// TIA Portal project "ScambioFerroviario" (V15.1)

(* hardware
DEVICE "S7-1200 station_1"  S7-1200 Station
   slot 0: "Telaio di montaggio_0"  S7-1200 Rack  Rack  V1.0
   slot 1: "PLC_1"  CPU 1214C DC/DC/DC  6ES7 214-1AG40-0XB0  V4.2
*)

// ===== PLC "PLC_1"  CPU 1214C DC/DC/DC =====

VAR_GLOBAL   // PLC tag table "Tabella delle variabili standard"
   "Mutex" AT %M0.0 : Bool;
   "P1" AT %I0.0 : Bool;
   "P2" AT %I0.1 : Bool;
   "SP1" AT %I0.2 : Bool;
   "SP2" AT %I0.3 : Bool;
   "SA1" AT %I0.4 : Bool;
   "SA2" AT %I0.5 : Bool;
   "A" AT %I0.6 : Bool;
   "B" AT %I0.7 : Bool;
   "C" AT %I1.0 : Bool;
   "D" AT %I1.1 : Bool;
   "S1" AT %Q0.0 : Bool;
   "D1" AT %Q0.1 : Bool;
   "S2" AT %Q0.2 : Bool;
   "D2" AT %Q0.3 : Bool;
   "SC1" AT %Q0.4 : Bool;
   "SC2" AT %Q0.5 : Bool;
END_VAR

VAR_GLOBAL CONSTANT   // PLC tag table "Tabella delle variabili standard"
   "AttesaRifornimento" : Time := T#1m;
END_VAR

TYPE "StatoCorsaSingola"
   STRUCT
      Home : Bool := true;
      Checkpoint : Bool;
      AcquisisciLock : Bool;
      ZonaCritica : Bool;
      RilasciaLock : Bool;
      FineCorsa : Bool;
   END_STRUCT;
END_TYPE

DATA_BLOCK "AndataCarrello1_DB"   // DB1
{ S7_Optimized_Access := 'TRUE' }
VERSION : 0.1
// stored: InstanceOfName CorsaSingola
"CorsaSingola"
BEGIN
END_DATA_BLOCK

DATA_BLOCK "RitornoCarrello1_DB"   // DB2
{ S7_Optimized_Access := 'TRUE' }
VERSION : 0.1
// stored: InstanceOfName CorsaSingola
"CorsaSingola"
BEGIN
END_DATA_BLOCK

DATA_BLOCK "AndataCarrello2_DB"   // DB4
{ S7_Optimized_Access := 'TRUE' }
VERSION : 0.1
// stored: InstanceOfName CorsaSingola
"CorsaSingola"
BEGIN
END_DATA_BLOCK

DATA_BLOCK "RitornoCarrello2_DB"   // DB5
{ S7_Optimized_Access := 'TRUE' }
VERSION : 0.1
// stored: InstanceOfName CorsaSingola
"CorsaSingola"
BEGIN
END_DATA_BLOCK

// folder: System blocks/Program resources

DATA_BLOCK "IEC_Timer_0_DB"   // DB3
{ S7_Optimized_Access := 'TRUE' }
AUTHOR : Simatic
FAMILY : IEC
NAME : IEC_TMR
VERSION : 1.0
// stored: InstanceOfName IEC_TIMER
"IEC_TIMER"
BEGIN
END_DATA_BLOCK

DATA_BLOCK "IEC_Timer_1_DB"   // DB6
{ S7_Optimized_Access := 'TRUE' }
AUTHOR : Simatic
FAMILY : IEC
NAME : IEC_TMR
VERSION : 1.0
// stored: InstanceOfName IEC_TIMER
"IEC_TIMER"
BEGIN
END_DATA_BLOCK

// folder: (top level)

FUNCTION_BLOCK "CorsaSingola"   // FB1, LAD
{ S7_Optimized_Access := 'TRUE' }
VERSION : 0.1
   VAR_INPUT
      Abilita : Bool;
      SP : Bool;
      Fotocellula1 : Bool;
      Fotocellula2 : Bool;
      SA : Bool;
   END_VAR
   VAR_OUTPUT
      SC_0 : Bool;   // Passare qui lo scambio da settare a LOW
      SC_1 : Bool;   // Passare qui lo scambio da settare a HIGH
      "M" : Bool;
   END_VAR
   VAR_IN_OUT
      Mutex : Bool;
   END_VAR
   VAR RETAIN
      Stato : "StatoCorsaSingola";
   END_VAR
BEGIN

REGION Network 1
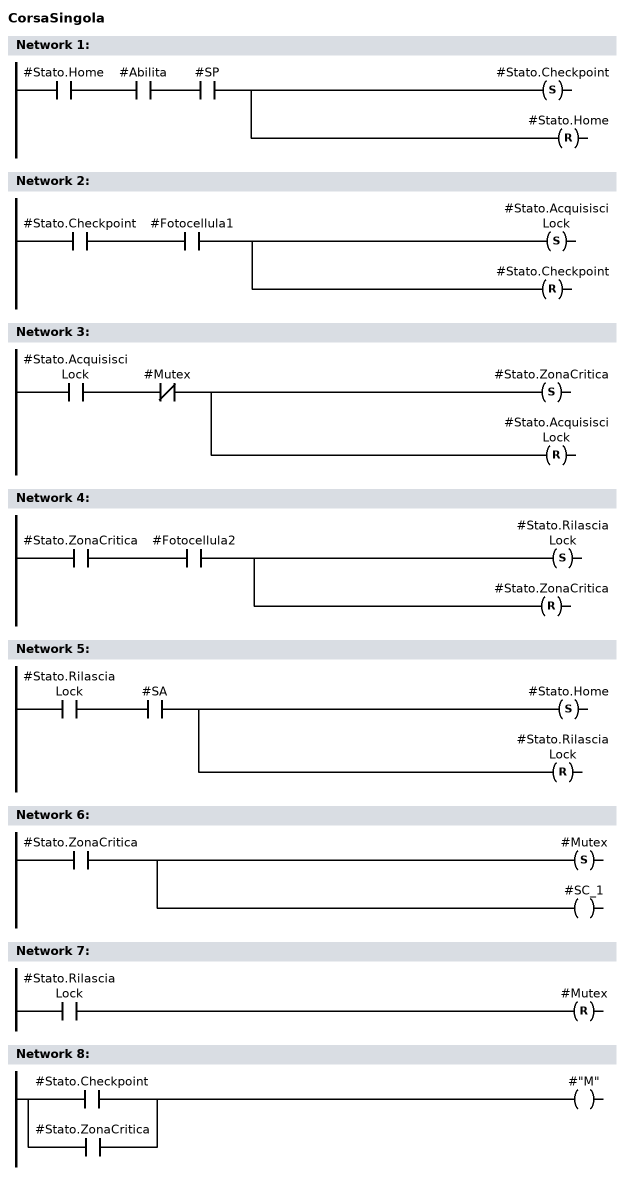
   RUNG wire#powerrail
      Contact( #Stato.Home )
      Contact( #Abilita )
      Contact( #SP )
      wire#w1
      S_Coil( #Stato.Checkpoint )
   END_RUNG
   RUNG wire#w1
      R_Coil( #Stato.Home )
   END_RUNG
   // the same network as SCL:
   IF #Stato.Home AND #Abilita AND #SP THEN
       #Stato.Checkpoint := TRUE;
       #Stato.Home := FALSE;
   END_IF;
END_REGION

REGION Network 2
   RUNG wire#powerrail
      Contact( #Stato.Checkpoint )
      Contact( #Fotocellula1 )
      wire#w1
      S_Coil( #Stato.AcquisisciLock )
   END_RUNG
   RUNG wire#w1
      R_Coil( #Stato.Checkpoint )
   END_RUNG
   // the same network as SCL:
   IF #Stato.Checkpoint AND #Fotocellula1 THEN
       #Stato.AcquisisciLock := TRUE;
       #Stato.Checkpoint := FALSE;
   END_IF;
END_REGION

REGION Network 3
   RUNG wire#powerrail
      Contact( #Stato.AcquisisciLock )
      I_Contact( #Mutex )
      wire#w1
      S_Coil( #Stato.ZonaCritica )
   END_RUNG
   RUNG wire#w1
      R_Coil( #Stato.AcquisisciLock )
   END_RUNG
   // the same network as SCL:
   IF #Stato.AcquisisciLock AND NOT #Mutex THEN
       #Stato.ZonaCritica := TRUE;
       #Stato.AcquisisciLock := FALSE;
   END_IF;
END_REGION

REGION Network 4
   RUNG wire#powerrail
      Contact( #Stato.ZonaCritica )
      Contact( #Fotocellula2 )
      wire#w1
      S_Coil( #Stato.RilasciaLock )
   END_RUNG
   RUNG wire#w1
      R_Coil( #Stato.ZonaCritica )
   END_RUNG
   // the same network as SCL:
   IF #Stato.ZonaCritica AND #Fotocellula2 THEN
       #Stato.RilasciaLock := TRUE;
       #Stato.ZonaCritica := FALSE;
   END_IF;
END_REGION

REGION Network 5
   RUNG wire#powerrail
      Contact( #Stato.RilasciaLock )
      Contact( #SA )
      wire#w1
      S_Coil( #Stato.Home )
   END_RUNG
   RUNG wire#w1
      R_Coil( #Stato.RilasciaLock )
   END_RUNG
   // the same network as SCL:
   IF #Stato.RilasciaLock AND #SA THEN
       #Stato.Home := TRUE;
       #Stato.RilasciaLock := FALSE;
   END_IF;
END_REGION

REGION Network 6
   RUNG wire#powerrail
      Contact( #Stato.ZonaCritica )
      wire#w1
      S_Coil( #Mutex )
   END_RUNG
   RUNG wire#w1
      Coil( #SC_1 )
   END_RUNG
   // the same network as SCL:
   IF #Stato.ZonaCritica THEN #Mutex := TRUE; END_IF;
   #SC_1 := #Stato.ZonaCritica;
END_REGION

REGION Network 7
   RUNG wire#powerrail
      Contact( #Stato.RilasciaLock )
      R_Coil( #Mutex )
   END_RUNG
   // the same network as SCL:
   IF #Stato.RilasciaLock THEN #Mutex := FALSE; END_IF;
END_REGION

REGION Network 8
   RUNG wire#powerrail
      Contact( #Stato.Checkpoint )
      wire#w1
      Coil( #"M" )
   END_RUNG
   RUNG wire#powerrail
      Contact( #Stato.ZonaCritica )
   END_RUNG wire#w1
   // the same network as SCL:
   #"M" := #Stato.Checkpoint OR #Stato.ZonaCritica;
END_REGION
END_FUNCTION_BLOCK

ORGANIZATION_BLOCK "Main"   // OB1, LAD, ProgramCycle
TITLE = "Main Program Sweep (Cycle)"
{ S7_Optimized_Access := 'TRUE' }
VERSION : 0.1
   VAR_INPUT
      Initial_Call : Bool;   // Initial call of this OB
      Remanence : Bool;   // =True, if remanent data are available
   END_VAR
BEGIN

REGION Network 1
   // Carrello1
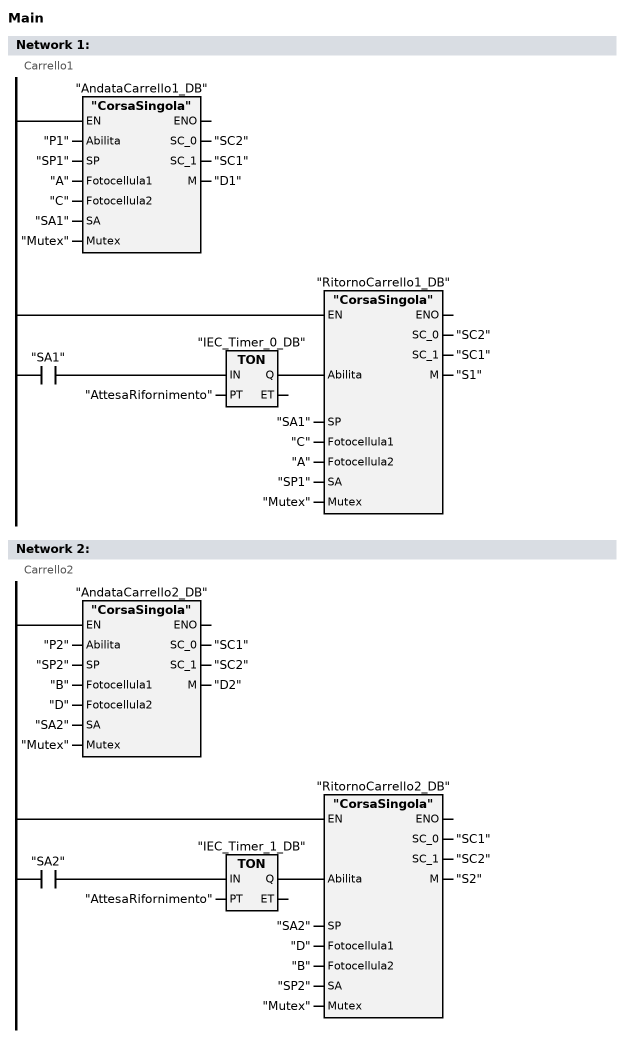
   "AndataCarrello1_DB"(Abilita := "P1",   // "CorsaSingola"
                        SP := "SP1",
                        Fotocellula1 := "A",
                        Fotocellula2 := "C",
                        SA := "SA1",
                        Mutex := "Mutex",
                        SC_0 => "SC2",
                        SC_1 => "SC1",
                        "M" => "D1");
   "IEC_Timer_0_DB".TON(IN := "SA1", PT := "AttesaRifornimento");
   "RitornoCarrello1_DB"(Abilita := "IEC_Timer_0_DB".Q,   // "CorsaSingola"
                         SP := "SA1",
                         Fotocellula1 := "C",
                         Fotocellula2 := "A",
                         SA := "SP1",
                         Mutex := "Mutex",
                         SC_0 => "SC2",
                         SC_1 => "SC1",
                         "M" => "S1");
END_REGION

REGION Network 2
   // Carrello2
   "AndataCarrello2_DB"(Abilita := "P2",   // "CorsaSingola"
                        SP := "SP2",
                        Fotocellula1 := "B",
                        Fotocellula2 := "D",
                        SA := "SA2",
                        Mutex := "Mutex",
                        SC_0 => "SC1",
                        SC_1 => "SC2",
                        "M" => "D2");
   "IEC_Timer_1_DB".TON(IN := "SA2", PT := "AttesaRifornimento");
   "RitornoCarrello2_DB"(Abilita := "IEC_Timer_1_DB".Q,   // "CorsaSingola"
                         SP := "SA2",
                         Fotocellula1 := "D",
                         Fotocellula2 := "B",
                         SA := "SP2",
                         Mutex := "Mutex",
                         SC_0 => "SC1",
                         SC_1 => "SC2",
                         "M" => "S2");
END_REGION
END_ORGANIZATION_BLOCK